INTERFACE ISelection

METHOD TargetConverter : INT
VAR_INPUT
	sTargetName : STRING;	
END_VAR
VAR_OUTPUT
	TargetConverter_output : INT;	
END_VAR
END_METHOD

END_INTERFACE

(* stored: Version 1.1.0.1, ProductVersion 3.1.4024.6
   Itf ISelection: Id {d9fef92d-4ab6-4909-a2ac-3643f05873d4}
   Method TargetConverter: Id {cb25618b-b1c9-46c2-a593-5cf4696a2dbd} *)
